Yaskawa INFORM job: -70_-90.JBI

/JOB
//NAME -70_-90
///FOLDERNAME OBROTNIK
//POS
///NPOS 0,0,1,0,0,0
///TOOL 0
///POSTYPE PULSE
///PULSE
EC00000=620788,1112951
//INST
///DATE 2023/11/07 18:52
///ATTR SC,RW,RJ
////FRAME ROBOT
///GROUP1 ST1
NOP
MOVJ EC00000 VJ=100.00
END
